# EPICS autosave request: utcaApp/Db/fofb_cc.req
$(P)$(R)$(FOFB_CC)CCEnable-Sel
$(P)$(R)$(FOFB_CC)BPMId-SP
$(P)$(R)$(FOFB_CC)TimeFrameLen-SP
